(* IEC 61131-3 sources: actuators/test, 15 files *)

(* ---- Await.st ---- *)
USING AxUnit.Assert;
USING Simatic.Ax.Commands;

NAMESPACE Simatic.Ax.Actuators

    // Helper function to await the completion of a command and return its state.
    FUNCTION Await : PlcOpen
        VAR_INPUT
            cmd : itfCommand;
        END_VAR

        IF (NOT cmd.Busy()) THEN
            IF cmd.Done() THEN
                Await := PlcOpen#Done;
                RETURN;
            ELSIF cmd.Error() THEN
                Await := PlcOpen#Error;
                RETURN;
            ELSIF cmd.CommandAborted() THEN
                Await := PlcOpen#Aborted;
                RETURN;
            ELSE
                Await := PlcOpen#Undefined;
                RETURN;
            END_IF;
        ELSE
            Await := PlcOpen#Busy;
            RETURN;
        END_IF;
    END_FUNCTION

    // Enumeration representing the possible states of a PLCOpen command.
    TYPE
        PlcOpen : (Busy, Done, Error, Aborted, Undefined) := Undefined;
    END_TYPE

END_NAMESPACE

(* ---- ActuatorStateAssertions.st ---- *)
USING System.Strings;
USING AxUnit.ResultFunctions;
USING Simatic.Ax.Actuators;

NAMESPACE AxUnit.Assert

    FUNCTION Equal
        VAR_INPUT
            expected : ActuatorState;
            actual : ActuatorState;
            {CallerFilePath}
            file : WSTRING[1024];
            {CallerLineNumber}
            line : INT;
        END_VAR
        VAR_TEMP
            messageStr : STRING;
        END_VAR

        IF expected = actual THEN
            axunit_Succeed();
        ELSE
            messageStr := Concat('Expected = ', Simatic.Ax.Actuators.ToString(val := expected), ' Actual = ', Simatic.Ax.Actuators.ToString(actual));
            axunit_Fail(messageStr, file, line);
        END_IF;
        AxUnit.Assert.Equal(expected := TRUE, actual := expected = actual);
        ;
    END_FUNCTION

    FUNCTION NotEqual
        VAR_INPUT
            expected : ActuatorState;
            actual : ActuatorState;
            {CallerFilePath}
            file : WSTRING[1024];
            {CallerLineNumber}
            line : INT;
        END_VAR
        VAR_TEMP
            messageStr : STRING;
        END_VAR
        IF expected = actual THEN
            axunit_Succeed();
        ELSE
            messageStr := Concat('Expected = ', Simatic.Ax.Actuators.ToString(expected), 'Actual = ', Simatic.Ax.Actuators.ToString(actual));
            axunit_Fail(messageStr, file, line);
        END_IF;
        AxUnit.Assert.Equal(expected := TRUE, actual := expected <> actual);
        ;
    END_FUNCTION

END_NAMESPACE

(* ---- Asserts.st ---- *)
USING System.Strings;
USING AxUnit.ResultFunctions;

NAMESPACE AxUnit.Assert

    FUNCTION Equal
        VAR_INPUT
            expected : STRING;
            actual : STRING;
            {CallerFilePath}
            file : WSTRING[1024];
            {CallerLineNumber}
            line : INT;
        END_VAR
        VAR_TEMP
            messageStr : STRING;
        END_VAR

        IF expected = actual THEN
            axunit_Succeed();
        ELSE
            messageStr := Concat('Expected = ', expected, 'Actual = ', actual);
            axunit_Fail(messageStr, file, line);
        END_IF;
        Equal(expected := TRUE, actual := expected = actual);
        ;
    END_FUNCTION

    FUNCTION NotEqual
        VAR_INPUT
            expected : STRING;
            actual : STRING;
            {CallerFilePath}
            file : WSTRING[1024];
            {CallerLineNumber}
            line : INT;
        END_VAR
        VAR_TEMP
            messageStr : STRING;
        END_VAR

        IF expected = actual THEN
            axunit_Succeed();
        ELSE
            messageStr := Concat('Expected = ', expected, 'Actual = ', actual);
            axunit_Fail(messageStr, file, line);
        END_IF;
        Equal(expected := TRUE, actual := expected <> actual);
        ;
    END_FUNCTION

END_NAMESPACE

(* ---- Boolean.st ---- *)
USING AxUnit.ResultFunctions;
USING System.Strings;

NAMESPACE AxUnit.Assert

    FUNCTION PUBLIC IsTrue
        VAR_INPUT
            condition : BOOL;

            {CallerFilePath}
            file : WSTRING[1024];
            {CallerLineNumber}
            line : INT;
        END_VAR

        IF condition THEN
            axunit_Succeed();
        ELSE
            axunit_Fail('Condition is not true', file, line);
        END_IF;

    END_FUNCTION

    FUNCTION PUBLIC IsFalse
        VAR_INPUT
            condition : BOOL;

            {CallerFilePath}
            file : WSTRING[1024];
            {CallerLineNumber}
            line : INT;
        END_VAR

        IF NOT condition THEN
            axunit_Succeed();
        ELSE
            axunit_Fail('Condition is not false', file, line);
        END_IF;

    END_FUNCTION

END_NAMESPACE

(* ---- PlcOpenAssert.st ---- *)
USING Simatic.Ax.Commands;
USING System.Strings;
USING AxUnit.ResultFunctions;

NAMESPACE AxUnit.Assert

    FUNCTION Equal
        VAR_INPUT
            expected : PlcOpen;
            actual : PlcOpen;
            {CallerFilePath}
            file : WSTRING[1024];
            {CallerLineNumber}
            line : INT;
        END_VAR
        VAR_TEMP
            messageStr : STRING;
        END_VAR

        IF expected = actual THEN
            axunit_Succeed();
        ELSE
            messageStr := Concat('Expected = ', ToString(expected), 'Actual = ', ToString(actual));
            axunit_Fail(messageStr, file, line);
        END_IF;
        Equal(expected := TRUE, actual := expected = actual);
        ;
    END_FUNCTION

    FUNCTION NotEqual
        VAR_INPUT
            expected : PlcOpen;
            actual : PlcOpen;
            {CallerFilePath}
            file : WSTRING[1024];
            {CallerLineNumber}
            line : INT;
        END_VAR
        VAR_TEMP
            messageStr : STRING;
        END_VAR

        IF expected = actual THEN
            axunit_Succeed();
        ELSE
            messageStr := Concat('Expected = ', ToString(expected), ' Actual = ', ToString(actual));
            axunit_Fail(messageStr, file, line);
        END_IF;
        Equal(expected := TRUE, actual := expected <> actual);
        ;
    END_FUNCTION

END_NAMESPACE

(* ---- EndSwitchMock.st ---- *)
USING AxUnit.Assert;

NAMESPACE Simatic.Ax.Actuators

    /// Mock implementation of an activated endswitch for testing purposes.
    /// Input: None.
    /// Returns: Always returns TRUE for IsActivated, FALSE for all other state queries.
    CLASS EndSwitchMockActivated IMPLEMENTS itfEndswitch

        /// Starts monitoring the endswitch with a specified monitoring time.
        /// Input: Mode - The supervision mode to enable.
        /// Returns: None.
        METHOD PUBLIC EnableSupervision
            VAR_INPUT
                Mode : SuperVisionMode;
            END_VAR

            ;
        END_METHOD

        /// Checks if the endswitch is currently activated.
        /// Input: None.
        /// Returns: Always TRUE to simulate an activated endswitch.
        METHOD PUBLIC IsActivated : BOOL
            IsActivated := TRUE;
            ;
        END_METHOD

        /// Checks if the endswitch has been reached.
        /// Input: None.
        /// Returns: Always FALSE for this mock.
        METHOD PUBLIC HasReached : BOOL
            HasReached := FALSE;
            ;
        END_METHOD

        /// Checks if the endswitch has been left.
        /// Input: None.
        /// Returns: Always FALSE for this mock.
        METHOD PUBLIC HasLeft : BOOL
            HasLeft := FALSE;
            ;
        END_METHOD

        /// Checks if the monitoring time has elapsed.
        /// Input: None.
        /// Returns: Always FALSE for this mock.
        METHOD PUBLIC TimeHasElapsed : BOOL
            TimeHasElapsed := FALSE;
        END_METHOD

        /// Returns the error status of the endswitch.
        /// Input: None.
        /// Returns: Default supervision error state.
        METHOD PUBLIC GetError : SuperVisionState
            ;
        END_METHOD
    END_CLASS

    /// Mock implementation of an endswitch that has been reached for testing purposes.
    /// Input: None.
    /// Returns: TRUE for IsActivated and HasReached, FALSE for other state queries.
    CLASS EndSwitchMockHasReached IMPLEMENTS itfEndswitch

        /// Starts monitoring the endswitch with a specified monitoring time.
        /// Input: Mode - The supervision mode to enable.
        /// Returns: None.
        METHOD PUBLIC EnableSupervision
            VAR_INPUT
                Mode : SuperVisionMode;
            END_VAR
            ;
        END_METHOD

        /// Checks if the endswitch is currently activated.
        /// Input: None.
        /// Returns: Always TRUE to simulate an activated endswitch.
        METHOD PUBLIC IsActivated : BOOL
            IsActivated := TRUE;
            ;
        END_METHOD

        /// Checks if the endswitch has been reached.
        /// Input: None.
        /// Returns: Always TRUE to simulate a reached endswitch.
        METHOD PUBLIC HasReached : BOOL
            HasReached := TRUE;
            ;
        END_METHOD

        /// Checks if the endswitch has been left.
        /// Input: None.
        /// Returns: Always FALSE for this mock.
        METHOD PUBLIC HasLeft : BOOL
            HasLeft := FALSE;
            ;
        END_METHOD

        /// Checks if the monitoring time has elapsed.
        /// Input: None.
        /// Returns: Always FALSE for this mock.
        METHOD PUBLIC TimeHasElapsed : BOOL
            TimeHasElapsed := FALSE;
        END_METHOD

        /// Returns the error status of the endswitch.
        /// Input: None.
        /// Returns: Default supervision error state.
        METHOD PUBLIC GetError : SuperVisionState
            ;
        END_METHOD
    END_CLASS

    /// Mock implementation of an endswitch that has been left for testing purposes.
    /// Input: None.
    /// Returns: TRUE for HasLeft, FALSE for other state queries.
    CLASS EndSwitchMockHasLeft IMPLEMENTS itfEndswitch

        /// Starts monitoring the endswitch with a specified monitoring time.
        /// Input: Mode - The supervision mode to enable.
        /// Returns: None.
        METHOD PUBLIC EnableSupervision
            VAR_INPUT
                Mode : SuperVisionMode;
            END_VAR

            ;
        END_METHOD

        /// Checks if the endswitch is currently activated.
        /// Input: None.
        /// Returns: Always FALSE to simulate a deactivated endswitch.
        METHOD PUBLIC IsActivated : BOOL
            IsActivated := FALSE;
            ;
        END_METHOD

        /// Checks if the endswitch has been reached.
        /// Input: None.
        /// Returns: Always FALSE for this mock.
        METHOD PUBLIC HasReached : BOOL
            HasReached := FALSE;
            ;
        END_METHOD

        /// Checks if the endswitch has been left.
        /// Input: None.
        /// Returns: Always TRUE to simulate a left endswitch.
        METHOD PUBLIC HasLeft : BOOL
            HasLeft := TRUE;
            ;
        END_METHOD

        /// Checks if the monitoring time has elapsed.
        /// Input: None.
        /// Returns: Always FALSE for this mock.
        METHOD PUBLIC TimeHasElapsed : BOOL
            TimeHasElapsed := FALSE;
        END_METHOD

        /// Returns the error status of the endswitch.
        /// Input: None.
        /// Returns: Default supervision error state.
        METHOD PUBLIC GetError : SuperVisionState
            ;
        END_METHOD
    END_CLASS

    /// Mock implementation of a non-activated endswitch for testing purposes.
    /// Input: None.
    /// Returns: FALSE for all state queries to simulate an inactive endswitch.
    CLASS EndSwitchMockNotActivated IMPLEMENTS itfEndswitch

        /// Starts monitoring the endswitch with a specified monitoring time.
        /// Input: Mode - The supervision mode to enable.
        /// Returns: None.
        METHOD PUBLIC EnableSupervision
            VAR_INPUT
                Mode : SuperVisionMode;
            END_VAR

            ;
        END_METHOD

        /// Disables monitoring of the endswitch.
        /// Input: None.
        /// Returns: None.
        METHOD PUBLIC DisableMonitoring
            ;
        END_METHOD

        /// Checks if the endswitch is currently activated.
        /// Input: None.
        /// Returns: Always FALSE to simulate an inactive endswitch.
        METHOD PUBLIC IsActivated : BOOL
            IsActivated := FALSE;
            ;
        END_METHOD

        /// Checks if the endswitch has been reached.
        /// Input: None.
        /// Returns: Always FALSE for this mock.
        METHOD PUBLIC HasReached : BOOL
            HasReached := FALSE;
            ;
        END_METHOD

        /// Checks if the endswitch has been left.
        /// Input: None.
        /// Returns: Always FALSE for this mock.
        METHOD PUBLIC HasLeft : BOOL
            HasLeft := FALSE;
            ;
        END_METHOD

        /// Checks if the monitoring time has elapsed.
        /// Input: None.
        /// Returns: Always FALSE for this mock.
        METHOD PUBLIC TimeHasElapsed : BOOL
            TimeHasElapsed := FALSE;
        END_METHOD

        /// Returns the error status of the endswitch.
        /// Input: None.
        /// Returns: Default supervision error state.
        METHOD PUBLIC GetError : SuperVisionState
            ;
        END_METHOD
    END_CLASS
END_NAMESPACE

(* ---- TestActuator2Way.st ---- *)
USING AxUnit.Assert;
USING Simatic.Ax.Commands;

NAMESPACE Simatic.Ax.Actuators

    {TestFixture}
    // Test class for the Actuator2Way class.
    // This class contains tests to verify the behavior of the Actuator2Way component.
    CLASS TestActuator2Way
        VAR
            // Instance of Actuator2Way for testing.
            _actuator, _actuatorStateless : Actuator2Way;

            // Command interface for actuator operations.
            _cmd : itfCommand;

            // State of the PLCOpen command.
            _plcOpenState : PlcOpen;

            // Mock sensors for testing actuator behavior.
            _sensorActivated : EndSwitchMockActivated;
            _sensorNotActivated : EndSwitchMockNotActivated;
            _sensorHasReached : EndSwitchMockHasReached;
            _sensorHasLeft : EndSwitchMockHasLeft;

            // Actuator Controls
            ActuatorMoveToHomePos : PositionControl;
            ActuatorMoveToWorkPos : PositionControl;
        END_VAR

        {TestSetup}
        // Sets up the test environment by initializing the actuator instance and assigning mock sensors and controls.
        METHOD PUBLIC Setup
            _actuator := _actuatorStateless;
            _actuator.Q_ToHomePosition := ActuatorMoveToHomePos;
            _actuator.Q_ToWorkPosition := ActuatorMoveToWorkPos;
        END_METHOD

        {Test}
        // Verifies that the initial state of the actuator is Undefined.
        METHOD PUBLIC TestInitialState
            VAR
                initialState : ActuatorState;
            END_VAR

            // Step 1: Retrieve the initial state of the actuator.
            initialState := _actuator.GetState();

            // Step 2: Assert that the initial state is Undefined.
            Equal(expected := ActuatorState#Undefined, actual := initialState);
        END_METHOD

        {Test}
        // Tests the transition to MoveToWorkPosition state when not in the work position.
        METHOD PUBLIC Command_MoveToWorkPosition_Returns_State_MoveToWorkPosition_When_NotInWorkpos
            VAR
                resultHome, resultWork : BOOL;
            END_VAR

            // Step 1: Set initial sensor states to indicate the actuator is not in any position.
            _actuator.I_InHomePosition := _sensorNotActivated;
            _actuator.I_InWorkPosition := _sensorNotActivated;

            // Step 2: Issue the command to move to work position.
            _cmd := _actuator.GoToWorkPosition();
            _plcOpenState := Await(_cmd);

            // Step 3: Verify the actuator is in the MoveToWorkPosition state.
            Equal(expected := PlcOpen#Busy, actual := _plcOpenState);
            Equal(expected := ActuatorState#MoveToWorkPosition, actual := _actuator.GetState());

            // Step 4: Check the actuator outputs.
            ActuatorMoveToHomePos.WriteCyclic(Q => resultHome);
            ActuatorMoveToWorkPos.WriteCyclic(Q => resultWork);
            IsFalse(condition := resultHome);
            IsTrue(condition := resultWork);

            // Step 5: Simulate reaching the work position.
            _actuator.I_InWorkPosition := _sensorHasReached;
            _plcOpenState := Await(_cmd);

            // Step 6: Verify the actuator has reached the work position.
            Equal(expected := PlcOpen#Done, actual := _plcOpenState);
            Equal(expected := ActuatorState#InWorkPosition, actual := _actuator.GetState());

            // Step 7: Check the actuator outputs again.
            ActuatorMoveToHomePos.WriteCyclic(Q => resultHome);
            ActuatorMoveToWorkPos.WriteCyclic(Q => resultWork);
            IsFalse(condition := resultHome);
            IsFalse(condition := resultWork);
        END_METHOD

        {Test}
        // Tests that the actuator remains in InWorkPosition state when already in the work position.
        METHOD PUBLIC Command_MoveToWorkPosition_Returns_State_InWorkPosition_When_InWorkpos
            VAR
                isInWorkPos : BOOL := TRUE;
            END_VAR

            // Step 1: Set initial sensor states to indicate the actuator is already in the work position.
            _actuator.I_InHomePosition := _sensorNotActivated;
            _actuator.I_InWorkPosition := _sensorActivated;

            // Step 2: Issue the command to move to work position.
            _cmd := _actuator.GoToWorkPosition();
            _plcOpenState := Await(_cmd);

            // Step 3: Verify the actuator remains in the InWorkPosition state.
            Equal(expected := PlcOpen#Done, actual := _plcOpenState);
            Equal(expected := ActuatorState#InWorkPosition, actual := _actuator.GetState());
        END_METHOD

        {Test}
        // Tests the transition to MoveToHomePosition state when not in the home position.
        METHOD PUBLIC Command_MoveToHomePosition_Returns_State_MoveToHomePosition_When_NotIn_HomePos
            VAR
                resultHome, resultWork : BOOL;
            END_VAR

            // Step 1: Set initial sensor states to indicate the actuator is not in any position.
            _actuator.I_InHomePosition := _sensorNotActivated;
            _actuator.I_InWorkPosition := _sensorNotActivated;

            // Step 2: Issue the command to move to home position.
            _cmd := _actuator.GoToHomePosition();
            _plcOpenState := Await(_cmd);

            // Step 3: Verify the actuator is in the MoveToHomePosition state.
            Equal(expected := PlcOpen#Busy, actual := _plcOpenState);
            Equal(expected := ActuatorState#MoveToHomePosition, actual := _actuator.GetState());

            // Step 4: Check the actuator outputs.
            ActuatorMoveToHomePos.WriteCyclic(Q => resultHome);
            ActuatorMoveToWorkPos.WriteCyclic(Q => resultWork);
            IsTrue(condition := resultHome);
            IsFalse(condition := resultWork);

            // Step 5: Simulate reaching the home position.
            _actuator.I_InHomePosition := _sensorHasReached;
            _plcOpenState := Await(_cmd);

            // Step 6: Verify the actuator has reached the home position.
            Equal(expected := PlcOpen#Done, actual := _plcOpenState);
            Equal(expected := ActuatorState#InHomePosition, actual := _actuator.GetState());

            // Step 7: Check the actuator outputs again.
            ActuatorMoveToHomePos.WriteCyclic(Q => resultHome);
            ActuatorMoveToWorkPos.WriteCyclic(Q => resultWork);
            IsFalse(condition := resultHome);
            IsFalse(condition := resultWork);
        END_METHOD

        {Test}
        // Tests that the actuator remains in InHomePosition state when already in the home position.
        METHOD PUBLIC Command_MoveToHomePosition_Returns_State_InHomePosition_When_In_HomePos
            VAR
                isInHomePos : BOOL := TRUE;
            END_VAR

            // Step 1: Set initial sensor states to indicate the actuator is already in the home position.
            _actuator.I_InHomePosition := _sensorActivated;
            _actuator.I_InWorkPosition := _sensorNotActivated;

            // Step 2: Issue the command to move to home position.
            _cmd := _actuator.GoToHomePosition();
            _plcOpenState := Await(_cmd);

            // Step 3: Verify the actuator remains in the InHomePosition state.
            Equal(expected := PlcOpen#Done, actual := _plcOpenState);
            Equal(expected := ActuatorState#InHomePosition, actual := _actuator.GetState());
        END_METHOD

        {Test}
        // Tests multiple calls to the MoveToWorkPosition command.
        METHOD PUBLIC Call_Command_MoveToWorkPosition_Multiple
            VAR
                isInHomePos : BOOL := TRUE;
            END_VAR

            // Step 1: Set initial sensor states to indicate the actuator is not in any position.
            _actuator.I_InHomePosition := _sensorNotActivated;
            _actuator.I_InWorkPosition := _sensorNotActivated;

            // Step 2: Issue the command to move to work position multiple times.
            _cmd := _actuator.GoToWorkPosition();
            _plcOpenState := Await(_cmd);
            Equal(expected := PlcOpen#Busy, actual := _plcOpenState);
            Equal(expected := ActuatorState#MoveToWorkPosition, actual := _actuator.GetState());

            _cmd := _actuator.GoToWorkPosition();
            _plcOpenState := Await(_cmd);
            Equal(expected := PlcOpen#Busy, actual := _plcOpenState);
            Equal(expected := ActuatorState#MoveToWorkPosition, actual := _actuator.GetState());

            _cmd := _actuator.GoToWorkPosition();
            _plcOpenState := Await(_cmd);
            Equal(expected := PlcOpen#Busy, actual := _plcOpenState);
            Equal(expected := ActuatorState#MoveToWorkPosition, actual := _actuator.GetState());

            // Step 3: Simulate reaching the work position.
            _actuator.I_InWorkPosition := _sensorActivated;
            _cmd := _actuator.GoToWorkPosition();
            Equal(expected := ActuatorState#InWorkPosition, actual := _actuator.GetState());
            _plcOpenState := Await(_cmd);
            Equal(expected := PlcOpen#Done, actual := _plcOpenState);
            Equal(expected := ActuatorState#InWorkPosition, actual := _actuator.GetState());
        END_METHOD

        {Test}
        // Tests the behavior when MoveToWorkPosition is interrupted by MoveToHomePosition.
        METHOD PUBLIC Command_MoveToWorkPosition_Interrupted_By_MoveToHomePosition
            VAR
                resultHome, resultWork : BOOL;
            END_VAR

            // Step 1: Set initial sensor states to indicate the actuator is not in any position.
            _actuator.I_InHomePosition := _sensorNotActivated;
            _actuator.I_InWorkPosition := _sensorNotActivated;

            // Step 2: Start MoveToWorkPosition.
            _cmd := _actuator.GoToWorkPosition();
            _plcOpenState := Await(_cmd);

            // Step 3: Verify the actuator is in the MoveToWorkPosition state.
            Equal(expected := PlcOpen#Busy, actual := _plcOpenState);
            Equal(expected := ActuatorState#MoveToWorkPosition, actual := _actuator.GetState());

            // Step 4: Check the actuator outputs.
            ActuatorMoveToHomePos.WriteCyclic(Q => resultHome);
            ActuatorMoveToWorkPos.WriteCyclic(Q => resultWork);
            IsFalse(condition := resultHome);
            IsTrue(condition := resultWork);

            // Step 5: Interrupt with MoveToHomePosition.
            _cmd := _actuator.GoToHomePosition();
            _plcOpenState := Await(_cmd);

            // Step 6: Verify the actuator is in the MoveToHomePosition state.
            Equal(expected := PlcOpen#Busy, actual := _plcOpenState);
            Equal(expected := ActuatorState#MoveToHomePosition, actual := _actuator.GetState());

            // Step 7: Check the actuator outputs.
            ActuatorMoveToHomePos.WriteCyclic(Q => resultHome);
            ActuatorMoveToWorkPos.WriteCyclic(Q => resultWork);
            IsTrue(condition := resultHome);
            IsFalse(condition := resultWork);

            // Step 8: Simulate reaching the home position.
            _actuator.I_InHomePosition := _sensorHasReached;
            _plcOpenState := Await(_cmd);

            // Step 9: Verify the actuator has reached the home position.
            Equal(expected := PlcOpen#Done, actual := _plcOpenState);
            Equal(expected := ActuatorState#InHomePosition, actual := _actuator.GetState());

            // Step 10: Check the actuator outputs again.
            ActuatorMoveToHomePos.WriteCyclic(Q => resultHome);
            ActuatorMoveToWorkPos.WriteCyclic(Q => resultWork);
            IsFalse(condition := resultHome);
            IsFalse(condition := resultWork);
        END_METHOD

        {Test}
        // Tests the behavior when MoveToHomePosition is interrupted by MoveToWorkPosition.
        METHOD PUBLIC Command_MoveToHomePosition_Interrupted_By_MoveToWorkPosition
            VAR
                resultHome, resultWork : BOOL;
            END_VAR

            // Step 1: Set initial sensor states to indicate the actuator is not in any position.
            _actuator.I_InHomePosition := _sensorNotActivated;
            _actuator.I_InWorkPosition := _sensorNotActivated;

            // Step 2: Start MoveToHomePosition.
            _cmd := _actuator.GoToHomePosition();
            _plcOpenState := Await(_cmd);

            // Step 3: Verify the actuator is in the MoveToHomePosition state.
            Equal(expected := PlcOpen#Busy, actual := _plcOpenState);
            Equal(expected := ActuatorState#MoveToHomePosition, actual := _actuator.GetState());

            // Step 4: Check the actuator outputs.
            ActuatorMoveToHomePos.WriteCyclic(Q => resultHome);
            ActuatorMoveToWorkPos.WriteCyclic(Q => resultWork);
            IsTrue(condition := resultHome);
            IsFalse(condition := resultWork);

            // Step 5: Interrupt with MoveToWorkPosition.
            _cmd := _actuator.GoToWorkPosition();
            _plcOpenState := Await(_cmd);

            // Step 6: Verify the actuator is in the MoveToWorkPosition state.
            Equal(expected := PlcOpen#Busy, actual := _plcOpenState);
            Equal(expected := ActuatorState#MoveToWorkPosition, actual := _actuator.GetState());

            // Step 7: Check the actuator outputs.
            ActuatorMoveToHomePos.WriteCyclic(Q => resultHome);
            ActuatorMoveToWorkPos.WriteCyclic(Q => resultWork);
            IsFalse(condition := resultHome);
            IsTrue(condition := resultWork);

            // Step 8: Simulate reaching the work position.
            _actuator.I_InWorkPosition := _sensorHasReached;
            _plcOpenState := Await(_cmd);

            // Step 9: Verify the actuator has reached the work position.
            Equal(expected := PlcOpen#Done, actual := _plcOpenState);
            Equal(expected := ActuatorState#InWorkPosition, actual := _actuator.GetState());

            // Step 10: Check the actuator outputs again.
            ActuatorMoveToHomePos.WriteCyclic(Q => resultHome);
            ActuatorMoveToWorkPos.WriteCyclic(Q => resultWork);
            IsFalse(condition := resultHome);
            IsFalse(condition := resultWork);
        END_METHOD
    END_CLASS

END_NAMESPACE

(* ---- TestActuator2WayErrorHandling.st ---- *)
USING AxUnit.Assert;
USING Simatic.Ax.Commands;

NAMESPACE Simatic.Ax.Actuators

    {TestFixture}
    // Test class for the Actuator2Way class.
    // This class contains tests to verify the behavior of the Actuator2Way component.
    CLASS TestActuator2WayErrorHandling
        VAR
            // Instance of Actuator2Way for testing.
            _actuator, _actuatorStateless : Actuator2Way;

            // Command interface for actuator operations.
            _cmd : itfCommand;

            // State of the PLCOpen command.
            _plcOpenState : PlcOpen;

            // Mock sensors for testing actuator behavior.
            _sensorActivated : EndSwitchMockActivated;
            _sensorNotActivated : EndSwitchMockNotActivated;
            _sensorHasReached : EndSwitchMockHasReached;
            _sensorHasLeft : EndSwitchMockHasLeft;
            _sensorTimeHasElapsed : EndSwitchMockTimeHasElapsed;

            // Actuator Controls
            ActuatorMoveToHomePos : PositionControl;
            ActuatorMoveToWorkPos : PositionControl;
        END_VAR

        {TestSetup}
        // Sets up the test environment by initializing the actuator instance and assigning mock sensors and controls.
        METHOD PUBLIC Setup
            _actuator := _actuatorStateless;
            _actuator.Q_ToHomePosition := ActuatorMoveToHomePos;
            _actuator.Q_ToWorkPosition := ActuatorMoveToWorkPos;
            _actuator.I_InWorkPosition := _sensorNotActivated;
            _actuator.I_InHomePosition := _sensorNotActivated;
        END_METHOD

        {Test}
        // Tests the transition to MoveToWorkPosition state when not in the work position.
        METHOD PUBLIC Command_MoveToWorkPosition_Error_When_Sensor_Time_Has_Elapsed
            VAR
                resultHome, resultWork : BOOL;
            END_VAR

            // Step 1: Set initial sensor states to indicate the actuator is not in any position.
            _actuator.I_InHomePosition := _sensorNotActivated;
            _actuator.I_InWorkPosition := _sensorNotActivated;

            // Step 2: Issue the command to move to work position.
            _cmd := _actuator.GoToWorkPosition();
            _plcOpenState := Await(_cmd);

            // Step 3: Verify the actuator is in the MoveToWorkPosition state.
            Equal(expected := PlcOpen#Busy, actual := _plcOpenState);
            Equal(expected := ActuatorState#MoveToWorkPosition, actual := _actuator.GetState());

            // Step 4: Check the actuator outputs.
            ActuatorMoveToHomePos.WriteCyclic(Q => resultHome);
            ActuatorMoveToWorkPos.WriteCyclic(Q => resultWork);
            IsFalse(condition := resultHome);
            IsTrue(condition := resultWork);

            // Step 5: Simulate reaching the work position.
            _actuator.I_InWorkPosition := _sensorTimeHasElapsed;
            _plcOpenState := Await(_cmd);

            // Step 6: Verify the actuator has reached the work position.
            Equal(expected := PlcOpen#Error, actual := _plcOpenState);
            Equal(expected := ActuatorState#Error, actual := _actuator.GetState());

            // Step 7: Check the actuator outputs again.
            ActuatorMoveToHomePos.WriteCyclic(Q => resultHome);
            ActuatorMoveToWorkPos.WriteCyclic(Q => resultWork);
            IsFalse(condition := resultHome);
            IsFalse(condition := resultWork);
        END_METHOD

        {Test}
        // Tests the transition to MoveToHomePosition state when not in the home position.
        METHOD PUBLIC Reset_Actuator_Returns
            VAR
                resultHome, resultWork : BOOL;
            END_VAR
            THIS.Command_MoveToWorkPosition_Error_When_Sensor_Time_Has_Elapsed();
            // Step 1: Reset Actuator

            _actuator.Reset();

            // Step 2: Verify the actuator is in the MoveToHomePosition state.
            Equal(expected := ActuatorState#Undefined, actual := _actuator.GetState());

            // Step 3: Check the actuator outputs again.
            ActuatorMoveToHomePos.WriteCyclic(Q => resultHome);
            ActuatorMoveToWorkPos.WriteCyclic(Q => resultWork);
            IsFalse(condition := resultHome);
            IsFalse(condition := resultWork);
        END_METHOD

        {Test}
        // Tests the transition to MoveToWorkPosition state when not in the work position.
        METHOD PUBLIC Both_sensors_Active_Retrurs_Error
            VAR
                resultHome, resultWork : BOOL;
            END_VAR

            // Step 1: Set initial sensor states to indicate the actuator is not in any position.
            _actuator.I_InHomePosition := _sensorActivated;
            _actuator.I_InWorkPosition := _sensorActivated;

            // Step 2: Issue the command to move to work position.
            _cmd := _actuator.GoToWorkPosition();
            _plcOpenState := Await(_cmd);

            // Step 3: Verify the actuator is in the MoveToWorkPosition state.
            Equal(expected := PlcOpen#Error, actual := _plcOpenState);
            Equal(expected := ActuatorState#Error, actual := _actuator.GetState());

            // Step 4: Check the actuator outputs again.
            ActuatorMoveToHomePos.WriteCyclic(Q => resultHome);
            ActuatorMoveToWorkPos.WriteCyclic(Q => resultWork);
            IsFalse(condition := resultHome);
            IsFalse(condition := resultWork);
        END_METHOD
    END_CLASS

END_NAMESPACE

(* ---- TestActuator2WayWithLogger.st ---- *)
USING AxUnit.Assert;
USING Simatic.Ax.Commands;

NAMESPACE Simatic.Ax.Actuators

    {TestFixture}
    // Test class for the Actuator2Way class.
    // This class contains tests to verify the behavior of the Actuator2Way component.
    CLASS TestActuator2WayWithLogger
        VAR
            // Instance of Actuator2Way for testing.
            _actuator, _actuatorStateless : Actuator2Way;

            // Command interface for actuator operations.
            _cmd : itfCommand;

            // Logger
            _logger : StateLogger;
            _msgBuffer : ARRAY[1..1] OF LogMessage;

            // State of the PLCOpen command.
            _plcOpenState : PlcOpen;

            // Mock sensors for testing actuator behavior.
            _sensorActivated : EndSwitchMockActivated;
            _sensorNotActivated : EndSwitchMockNotActivated;
            _sensorHasReached : EndSwitchMockHasReached;
            _sensorHasLeft : EndSwitchMockHasLeft;

        END_VAR

        {TestSetup}
        // Sets up the test environment by initializing the actuator instance and assigning mock sensors and controls.
        METHOD PUBLIC Setup
            _actuator := _actuatorStateless;
            _actuator.Logger := _logger;
            _logger.MsgBuffer := REF(_msgBuffer);
            _logger.SetLogLevel(LogLevel#Info);
        END_METHOD

        {Test}
        // Tests the state transitions and verifies log entries in the StateLogger.
        METHOD PUBLIC Test_a_CompleteSequence_to_check_the_LogMessages
            VAR
                logEntry : STRING;
            END_VAR

            // Step 1: Set initial sensor states to indicate the actuator is in the home position.
            _actuator.I_InHomePosition := _sensorActivated;
            _actuator.I_InWorkPosition := _sensorNotActivated;

            // Step 2: Issue the command to move to work position.
            _cmd := _actuator.GoToWorkPosition();
            _plcOpenState := Await(_cmd);

            // Step 3: Verify the log entry for State changed to MoveToWorkPosition.
            logEntry := _logger.MsgBuffer^[1].message;
            Equal(expected := 'State changed to MoveToWorkPosition', actual := logEntry);

            // Step 4: Simulate reaching the work position.
            _actuator.I_InWorkPosition := _sensorHasReached;
            _actuator.I_InHomePosition := _sensorNotActivated;
            _plcOpenState := Await(_cmd);

            // Step 5: Verify the log entry for reaching InWorkPosition.
            logEntry := _logger.MsgBuffer^[1].message;
            Equal(expected := 'State changed to InWorkPosition', actual := logEntry);

            // Step 6: Issue the command to move to home position.
            _cmd := _actuator.GoToHomePosition();
            _plcOpenState := Await(_cmd);

            // Step 7: Verify the log entry for State changed to MoveToHomePosition.
            logEntry := _logger.MsgBuffer^[1].message;
            Equal(expected := 'State changed to MoveToHomePosition', actual := logEntry);

            // Step 8: Simulate reaching the home position.
            _actuator.I_InHomePosition := _sensorHasReached;
            _plcOpenState := Await(_cmd);

            // Step 9: Verify the log entry for reaching InHomePosition.
            logEntry := _logger.MsgBuffer^[1].message;
            Equal(expected := 'State changed to InHomePosition', actual := logEntry);
        END_METHOD

    END_CLASS

END_NAMESPACE

(* ---- TestActuator3Way.st ---- *)
USING AxUnit.Assert;
USING Simatic.Ax.Commands;

NAMESPACE Simatic.Ax.Actuators

    {TestFixture}
    // Test class for the Actuator3Way class.
    // This class contains tests to verify the behavior of the Actuator3Way component.
    CLASS TestActuator3Way
        VAR
            // Instance of Actuator3Way for testing.
            _actuator, _actuatorStateless : Actuator3Way;

            // Command interface for actuator operations.
            _cmd : itfCommand;

            // State of the PLCOpen command.
            _plcOpenState : PlcOpen;

            // Mock sensors for testing actuator behavior.
            _sensorActivated : EndSwitchMockActivated;
            _sensorNotActivated : EndSwitchMockNotActivated;
            _sensorHasReached : EndSwitchMockHasReached;
            _sensorHasLeft : EndSwitchMockHasLeft;

            // Actuator Controls
            ActuatorMoveToHomePos : PositionControl;
            ActuatorMoveToWorkPos : PositionControl;
            ActuatorMoveToWorkPos2 : PositionControl;
        END_VAR

        {TestSetup}
        // Sets up the test environment by initializing the actuator instance and assigning mock sensors and controls.
        METHOD PUBLIC Setup
            _actuator := _actuatorStateless;
            _actuator.Q_ToHomePosition := ActuatorMoveToHomePos;
            _actuator.Q_ToWorkPosition := ActuatorMoveToWorkPos;
            _actuator.Q_ToWorkPosition2 := ActuatorMoveToWorkPos2;
        END_METHOD

        {Test}
        // Verifies that the initial state of the actuator is Undefined.
        METHOD PUBLIC TestInitialState
            VAR
                initialState : ActuatorState;
            END_VAR

            // Step 1: Retrieve the initial state of the actuator.
            initialState := _actuator.GetState();

            // Step 2: Assert that the initial state is Undefined.
            Equal(expected := ActuatorState#Undefined, actual := initialState);
        END_METHOD

        {Test}
        // Tests the transition to MoveToWorkPosition state when not in the work position.
        METHOD PUBLIC Command_MoveToWorkPosition_Returns_State_MoveToWorkPosition_When_NotInWorkpos
            VAR
                resultHome, resultWork, resultWork2 : BOOL;
            END_VAR

            // Step 1: Set initial sensor states to indicate the actuator is not in any position.
            _actuator.I_InHomePosition := _sensorNotActivated;
            _actuator.I_InWorkPosition := _sensorNotActivated;
            _actuator.I_InWorkPosition2 := _sensorNotActivated;

            // Step 2: Issue the command to move to work position.
            _cmd := _actuator.GoToWorkPosition();
            _plcOpenState := Await(_cmd);

            // Step 3: Verify the actuator is in the MoveToWorkPosition state.
            AxUnit.Assert.Equal(expected := PlcOpen#Busy, actual := _plcOpenState);
            Equal(expected := ActuatorState#MoveToWorkPosition, actual := _actuator.GetState());

            // Step 4: Check the actuator outputs.
            ActuatorMoveToHomePos.WriteCyclic(Q => resultHome);
            ActuatorMoveToWorkPos.WriteCyclic(Q => resultWork);
            ActuatorMoveToWorkPos2.WriteCyclic(Q => resultWork2);
            IsFalse(condition := resultHome);
            IsTrue(condition := resultWork);
            IsFalse(condition := resultWork2);

            // Step 5: Simulate reaching the work position.
            _actuator.I_InWorkPosition := _sensorHasReached;
            _plcOpenState := Await(_cmd);

            // Step 6: Verify the actuator has reached the work position.
            AxUnit.Assert.Equal(expected := PlcOpen#Done, actual := _plcOpenState);
            Equal(expected := ActuatorState#InWorkPosition, actual := _actuator.GetState());

            // Step 7: Check the actuator outputs again.
            ActuatorMoveToHomePos.WriteCyclic(Q => resultHome);
            ActuatorMoveToWorkPos.WriteCyclic(Q => resultWork);
            ActuatorMoveToWorkPos2.WriteCyclic(Q => resultWork2);
            IsFalse(condition := resultHome);
            IsFalse(condition := resultWork);
            IsFalse(condition := resultWork2);
        END_METHOD

        {Test}
        // Tests the transition to MoveToWorkPosition2 state when not in the second work position.
        METHOD PUBLIC Command_MoveToWorkPosition2_Returns_State_MoveToWorkPosition2_When_NotInWorkpos2
            VAR
                resultHome, resultWork, resultWork2 : BOOL;
            END_VAR

            // Step 1: Set initial sensor states to indicate the actuator is not in any position.
            _actuator.I_InHomePosition := _sensorNotActivated;
            _actuator.I_InWorkPosition := _sensorNotActivated;
            _actuator.I_InWorkPosition2 := _sensorNotActivated;

            // Step 2: Issue the command to move to work position 2.
            _cmd := _actuator.GoToWorkPosition2();
            _plcOpenState := Await(_cmd);

            // Step 3: Verify the actuator is in the MoveToWorkPosition2 state.
            AxUnit.Assert.Equal(expected := PlcOpen#Busy, actual := _plcOpenState);
            Equal(expected := ActuatorState#MoveToWorkPosition2, actual := _actuator.GetState());

            // Step 4: Check the actuator outputs.
            ActuatorMoveToHomePos.WriteCyclic(Q => resultHome);
            ActuatorMoveToWorkPos.WriteCyclic(Q => resultWork);
            ActuatorMoveToWorkPos2.WriteCyclic(Q => resultWork2);
            IsFalse(condition := resultHome);
            IsFalse(condition := resultWork);
            IsTrue(condition := resultWork2);

            // Step 5: Simulate reaching the second work position.
            _actuator.I_InWorkPosition2 := _sensorHasReached;
            _plcOpenState := Await(_cmd);

            // Step 6: Verify the actuator has reached the second work position.
            AxUnit.Assert.Equal(expected := PlcOpen#Done, actual := _plcOpenState);
            Equal(expected := ActuatorState#InWorkPosition2, actual := _actuator.GetState());

            // Step 7: Check the actuator outputs again.
            ActuatorMoveToHomePos.WriteCyclic(Q => resultHome);
            ActuatorMoveToWorkPos.WriteCyclic(Q => resultWork);
            ActuatorMoveToWorkPos2.WriteCyclic(Q => resultWork2);
            IsFalse(condition := resultHome);
            IsFalse(condition := resultWork);
            IsFalse(condition := resultWork2);
        END_METHOD

        {Test}
        // Tests the transition to MoveToHomePosition state when not in the home position.
        METHOD PUBLIC Command_MoveToHomePosition_Returns_State_MoveToHomePosition_When_NotInHomePos
            VAR
                resultHome, resultWork, resultWork2 : BOOL;
            END_VAR

            // Step 1: Set initial sensor states to indicate the actuator is not in any position.
            _actuator.I_InHomePosition := _sensorNotActivated;
            _actuator.I_InWorkPosition := _sensorNotActivated;
            _actuator.I_InWorkPosition2 := _sensorNotActivated;

            // Step 2: Issue the command to move to home position.
            _cmd := _actuator.GoToHomePosition();
            _plcOpenState := Await(_cmd);

            // Step 3: Verify the actuator is in the MoveToHomePosition state.
            AxUnit.Assert.Equal(expected := PlcOpen#Busy, actual := _plcOpenState);
            Equal(expected := ActuatorState#MoveToHomePosition, actual := _actuator.GetState());

            // Step 4: Check the actuator outputs.
            ActuatorMoveToHomePos.WriteCyclic(Q => resultHome);
            ActuatorMoveToWorkPos.WriteCyclic(Q => resultWork);
            ActuatorMoveToWorkPos2.WriteCyclic(Q => resultWork2);
            IsTrue(condition := resultHome);
            IsFalse(condition := resultWork);
            IsFalse(condition := resultWork2);

            // Step 5: Simulate reaching the home position.
            _actuator.I_InHomePosition := _sensorHasReached;
            _plcOpenState := Await(_cmd);
            AxUnit.Assert.Equal(expected := PlcOpen#Done, actual := _plcOpenState);
            Equal(expected := ActuatorState#InHomePosition, actual := _actuator.GetState());

            ActuatorMoveToHomePos.WriteCyclic(Q => resultHome);
            ActuatorMoveToWorkPos.WriteCyclic(Q => resultWork);
            ActuatorMoveToWorkPos2.WriteCyclic(Q => resultWork2);
            IsFalse(condition := resultHome);
            IsFalse(condition := resultWork);
            IsFalse(condition := resultWork2);
        END_METHOD

        {Test}
        METHOD PUBLIC Call_Command_MoveToWorkPosition2_Multiple
            VAR
                isInHomePos : BOOL := TRUE;
            END_VAR

            _actuator.I_InHomePosition := _sensorNotActivated;
            _actuator.I_InWorkPosition := _sensorNotActivated;
            _actuator.I_InWorkPosition2 := _sensorNotActivated;

            _cmd := _actuator.GoToWorkPosition2();
            _plcOpenState := Await(_cmd);
            AxUnit.Assert.Equal(expected := PlcOpen#Busy, actual := _plcOpenState);
            Equal(expected := ActuatorState#MoveToWorkPosition2, actual := _actuator.GetState());

            _cmd := _actuator.GoToWorkPosition2();
            _plcOpenState := Await(_cmd);
            AxUnit.Assert.Equal(expected := PlcOpen#Busy, actual := _plcOpenState);
            Equal(expected := ActuatorState#MoveToWorkPosition2, actual := _actuator.GetState());

            _cmd := _actuator.GoToWorkPosition2();
            _plcOpenState := Await(_cmd);
            AxUnit.Assert.Equal(expected := PlcOpen#Busy, actual := _plcOpenState);
            Equal(expected := ActuatorState#MoveToWorkPosition2, actual := _actuator.GetState());

            _actuator.I_InWorkPosition2 := _sensorActivated;
            _cmd := _actuator.GoToWorkPosition2();
            Equal(expected := ActuatorState#InWorkPosition2, actual := _actuator.GetState());
            _plcOpenState := Await(_cmd);
            AxUnit.Assert.Equal(expected := PlcOpen#Done, actual := _plcOpenState);
            Equal(expected := ActuatorState#InWorkPosition2, actual := _actuator.GetState());
        END_METHOD

        {Test}
        METHOD PUBLIC Command_MoveToWorkPosition_Interrupted_By_MoveToHomePosition
            VAR
                resultHome, resultWork, resultWork2 : BOOL;
            END_VAR

            _actuator.I_InHomePosition := _sensorNotActivated;
            _actuator.I_InWorkPosition := _sensorNotActivated;
            _actuator.I_InWorkPosition2 := _sensorNotActivated;

            // Start MoveToWorkPosition
            _cmd := _actuator.GoToWorkPosition();
            _plcOpenState := Await(_cmd);

            AxUnit.Assert.Equal(expected := PlcOpen#Busy, actual := _plcOpenState);
            Equal(expected := ActuatorState#MoveToWorkPosition, actual := _actuator.GetState());

            ActuatorMoveToHomePos.WriteCyclic(Q => resultHome);
            ActuatorMoveToWorkPos.WriteCyclic(Q => resultWork);
            ActuatorMoveToWorkPos2.WriteCyclic(Q => resultWork2);
            IsFalse(condition := resultHome);
            IsTrue(condition := resultWork);
            IsFalse(condition := resultWork2);

            // Interrupt with MoveToHomePosition
            _cmd := _actuator.GoToHomePosition();
            _plcOpenState := Await(_cmd);

            AxUnit.Assert.Equal(expected := PlcOpen#Busy, actual := _plcOpenState);
            Equal(expected := ActuatorState#MoveToHomePosition, actual := _actuator.GetState());

            ActuatorMoveToHomePos.WriteCyclic(Q => resultHome);
            ActuatorMoveToWorkPos.WriteCyclic(Q => resultWork);
            ActuatorMoveToWorkPos2.WriteCyclic(Q => resultWork2);
            IsTrue(condition := resultHome);
            IsFalse(condition := resultWork);
            IsFalse(condition := resultWork2);

            _actuator.I_InHomePosition := _sensorHasReached;
            _plcOpenState := Await(_cmd);
            AxUnit.Assert.Equal(expected := PlcOpen#Done, actual := _plcOpenState);
            Equal(expected := ActuatorState#InHomePosition, actual := _actuator.GetState());

            // Step 7: Check the actuator outputs again.
            ActuatorMoveToHomePos.WriteCyclic(Q => resultHome);
            ActuatorMoveToWorkPos.WriteCyclic(Q => resultWork);
            ActuatorMoveToWorkPos2.WriteCyclic(Q => resultWork2);
            IsFalse(condition := resultHome);
            IsFalse(condition := resultWork);
            IsFalse(condition := resultWork2);
        END_METHOD

        {Test}
        METHOD PUBLIC Command_MoveToHomePosition_Interrupted_By_MoveToWorkPosition
            VAR
                resultHome, resultWork, resultWork2 : BOOL;
            END_VAR

            _actuator.I_InHomePosition := _sensorNotActivated;
            _actuator.I_InWorkPosition := _sensorNotActivated;
            _actuator.I_InWorkPosition2 := _sensorNotActivated;

            // Start MoveToHomePosition
            _cmd := _actuator.GoToHomePosition();
            _plcOpenState := Await(_cmd);

            AxUnit.Assert.Equal(expected := PlcOpen#Busy, actual := _plcOpenState);
            Equal(expected := ActuatorState#MoveToHomePosition, actual := _actuator.GetState());

            ActuatorMoveToHomePos.WriteCyclic(Q => resultHome);
            ActuatorMoveToWorkPos.WriteCyclic(Q => resultWork);
            ActuatorMoveToWorkPos2.WriteCyclic(Q => resultWork2);
            IsTrue(condition := resultHome);
            IsFalse(condition := resultWork);
            IsFalse(condition := resultWork2);

            // Interrupt with MoveToWorkPosition
            _cmd := _actuator.GoToWorkPosition();
            _plcOpenState := Await(_cmd);

            AxUnit.Assert.Equal(expected := PlcOpen#Busy, actual := _plcOpenState);
            Equal(expected := ActuatorState#MoveToWorkPosition, actual := _actuator.GetState());

            ActuatorMoveToHomePos.WriteCyclic(Q => resultHome);
            ActuatorMoveToWorkPos.WriteCyclic(Q => resultWork);
            ActuatorMoveToWorkPos2.WriteCyclic(Q => resultWork2);
            IsFalse(condition := resultHome);
            IsTrue(condition := resultWork);
            IsFalse(condition := resultWork2);

            _actuator.I_InWorkPosition := _sensorHasReached;
            _plcOpenState := Await(_cmd);
            AxUnit.Assert.Equal(expected := PlcOpen#Done, actual := _plcOpenState);
            Equal(expected := ActuatorState#InWorkPosition, actual := _actuator.GetState());

            ActuatorMoveToHomePos.WriteCyclic(Q => resultHome);
            ActuatorMoveToWorkPos.WriteCyclic(Q => resultWork);
            ActuatorMoveToWorkPos2.WriteCyclic(Q => resultWork2);
            IsFalse(condition := resultHome);
            IsFalse(condition := resultWork);
            IsFalse(condition := resultWork2);
        END_METHOD

        {Test}
        METHOD PUBLIC Command_MoveToWorkPosition2_Interrupted_By_MoveToHomePosition
            VAR
                resultHome, resultWork, resultWork2 : BOOL;
            END_VAR

            // Step 1: Set initial sensor states to indicate the actuator is not in any position.
            _actuator.I_InHomePosition := _sensorNotActivated;
            _actuator.I_InWorkPosition := _sensorNotActivated;
            _actuator.I_InWorkPosition2 := _sensorNotActivated;

            // Step 2: Start MoveToWorkPosition2.
            _cmd := _actuator.GoToWorkPosition2();
            _plcOpenState := Await(_cmd);

            // Step 3: Verify the actuator is in the MoveToWorkPosition2 state.
            AxUnit.Assert.Equal(expected := PlcOpen#Busy, actual := _plcOpenState);
            Equal(expected := ActuatorState#MoveToWorkPosition2, actual := _actuator.GetState());

            // Step 4: Check the actuator outputs.
            ActuatorMoveToHomePos.WriteCyclic(Q => resultHome);
            ActuatorMoveToWorkPos.WriteCyclic(Q => resultWork);
            ActuatorMoveToWorkPos2.WriteCyclic(Q => resultWork2);
            IsFalse(condition := resultHome);
            IsFalse(condition := resultWork);
            IsTrue(condition := resultWork2);

            // Step 5: Interrupt with MoveToHomePosition.
            _cmd := _actuator.GoToHomePosition();
            _plcOpenState := Await(_cmd);

            // Step 6: Verify the actuator is in the MoveToHomePosition state.
            AxUnit.Assert.Equal(expected := PlcOpen#Busy, actual := _plcOpenState);
            Equal(expected := ActuatorState#MoveToHomePosition, actual := _actuator.GetState());

            // Step 7: Check the actuator outputs.
            ActuatorMoveToHomePos.WriteCyclic(Q => resultHome);
            ActuatorMoveToWorkPos.WriteCyclic(Q => resultWork);
            ActuatorMoveToWorkPos2.WriteCyclic(Q => resultWork2);
            IsTrue(condition := resultHome);
            IsFalse(condition := resultWork);
            IsFalse(condition := resultWork2);

            // Step 8: Simulate reaching the home position.
            _actuator.I_InHomePosition := _sensorHasReached;
            _plcOpenState := Await(_cmd);

            // Step 9: Verify the actuator has reached the home position.
            AxUnit.Assert.Equal(expected := PlcOpen#Done, actual := _plcOpenState);
            Equal(expected := ActuatorState#InHomePosition, actual := _actuator.GetState());

            ActuatorMoveToHomePos.WriteCyclic(Q => resultHome);
            ActuatorMoveToWorkPos.WriteCyclic(Q => resultWork);
            ActuatorMoveToWorkPos2.WriteCyclic(Q => resultWork2);
            IsFalse(condition := resultHome);
            IsFalse(condition := resultWork);
            IsFalse(condition := resultWork2);
        END_METHOD

        {Test}
        METHOD PUBLIC Command_MoveToWorkPosition2_Interrupted_By_MoveToWorkPosition
            VAR
                resultHome, resultWork, resultWork2 : BOOL;
            END_VAR

            _actuator.I_InHomePosition := _sensorNotActivated;
            _actuator.I_InWorkPosition := _sensorNotActivated;
            _actuator.I_InWorkPosition2 := _sensorNotActivated;

            // Start MoveToWorkPosition2
            _cmd := _actuator.GoToWorkPosition2();
            _plcOpenState := Await(_cmd);

            AxUnit.Assert.Equal(expected := PlcOpen#Busy, actual := _plcOpenState);
            Equal(expected := ActuatorState#MoveToWorkPosition2, actual := _actuator.GetState());

            ActuatorMoveToHomePos.WriteCyclic(Q => resultHome);
            ActuatorMoveToWorkPos.WriteCyclic(Q => resultWork);
            ActuatorMoveToWorkPos2.WriteCyclic(Q => resultWork2);
            IsFalse(condition := resultHome);
            IsFalse(condition := resultWork);
            IsTrue(condition := resultWork2);

            // Interrupt with MoveToWorkPosition
            _cmd := _actuator.GoToWorkPosition();
            _plcOpenState := Await(_cmd);

            AxUnit.Assert.Equal(expected := PlcOpen#Busy, actual := _plcOpenState);
            Equal(expected := ActuatorState#MoveToWorkPosition, actual := _actuator.GetState());

            ActuatorMoveToHomePos.WriteCyclic(Q => resultHome);
            ActuatorMoveToWorkPos.WriteCyclic(Q => resultWork);
            ActuatorMoveToWorkPos2.WriteCyclic(Q => resultWork2);
            IsFalse(condition := resultHome);
            IsTrue(condition := resultWork);
            IsFalse(condition := resultWork2);

            _actuator.I_InWorkPosition := _sensorHasReached;
            _plcOpenState := Await(_cmd);
            AxUnit.Assert.Equal(expected := PlcOpen#Done, actual := _plcOpenState);
            Equal(expected := ActuatorState#InWorkPosition, actual := _actuator.GetState());

            ActuatorMoveToHomePos.WriteCyclic(Q => resultHome);
            ActuatorMoveToWorkPos.WriteCyclic(Q => resultWork);
            ActuatorMoveToWorkPos2.WriteCyclic(Q => resultWork2);
            IsFalse(condition := resultHome);
            IsFalse(condition := resultWork);
            IsFalse(condition := resultWork2);
        END_METHOD
    END_CLASS

END_NAMESPACE

(* ---- TestActuator3WayErrorHandling.st ---- *)
USING AxUnit.Assert;
USING Simatic.Ax.Commands;

NAMESPACE Simatic.Ax.Actuators

    {TestFixture}
    // Test class for the Actuator2Way class.
    // This class contains tests to verify the behavior of the Actuator2Way component.
    CLASS TestActuator3WayErrorHandling
        VAR
            // Instance of Actuator2Way for testing.
            _actuator, _actuatorStateless : Actuator3Way;

            // Command interface for actuator operations.
            _cmd : itfCommand;

            // State of the PLCOpen command.
            _plcOpenState : PlcOpen;

            // Mock sensors for testing actuator behavior.
            _sensorActivated : EndSwitchMockActivated;
            _sensorNotActivated : EndSwitchMockNotActivated;
            _sensorHasReached : EndSwitchMockHasReached;
            _sensorHasLeft : EndSwitchMockHasLeft;
            _sensorTimeHasElapsed : EndSwitchMockTimeHasElapsed;

            // Actuator Controls
            ActuatorMoveToHomePos : PositionControl;
            ActuatorMoveToWorkPos : PositionControl;
        END_VAR

        {TestSetup}
        // Sets up the test environment by initializing the actuator instance and assigning mock sensors and controls.
        METHOD PUBLIC Setup
            _actuator := _actuatorStateless;
            _actuator.Q_ToHomePosition := ActuatorMoveToHomePos;
            _actuator.Q_ToWorkPosition := ActuatorMoveToWorkPos;
            _actuator.I_InWorkPosition := _sensorNotActivated;
            _actuator.I_InHomePosition := _sensorNotActivated;
        END_METHOD

        {Test}
        // Tests the transition to MoveToWorkPosition state when not in the work position.
        METHOD PUBLIC Command_MoveToWorkPosition_Error_When_Sensor_Time_Has_Elapsed
            VAR
                resultHome, resultWork : BOOL;
            END_VAR

            // Step 1: Set initial sensor states to indicate the actuator is not in any position.
            _actuator.I_InHomePosition := _sensorNotActivated;
            _actuator.I_InWorkPosition := _sensorNotActivated;

            // Step 2: Issue the command to move to work position.
            _cmd := _actuator.GoToWorkPosition();
            _plcOpenState := Await(_cmd);

            // Step 3: Verify the actuator is in the MoveToWorkPosition state.
            Equal(expected := PlcOpen#Busy, actual := _plcOpenState);
            Equal(expected := ActuatorState#MoveToWorkPosition, actual := _actuator.GetState());

            // Step 4: Check the actuator outputs.
            ActuatorMoveToHomePos.WriteCyclic(Q => resultHome);
            ActuatorMoveToWorkPos.WriteCyclic(Q => resultWork);
            IsFalse(condition := resultHome);
            IsTrue(condition := resultWork);

            // Step 5: Simulate reaching the work position.
            _actuator.I_InWorkPosition := _sensorTimeHasElapsed;
            _plcOpenState := Await(_cmd);

            // Step 6: Verify the actuator has reached the work position.
            Equal(expected := PlcOpen#Error, actual := _plcOpenState);
            Equal(expected := ActuatorState#Error, actual := _actuator.GetState());

            // Step 7: Check the actuator outputs again.
            ActuatorMoveToHomePos.WriteCyclic(Q => resultHome);
            ActuatorMoveToWorkPos.WriteCyclic(Q => resultWork);
            IsFalse(condition := resultHome);
            IsFalse(condition := resultWork);
        END_METHOD

        {Test}
        // Tests the transition to MoveToHomePosition state when not in the home position.
        METHOD PUBLIC Reset_Actuator_Returns
            VAR
                resultHome, resultWork : BOOL;
            END_VAR
            THIS.Command_MoveToWorkPosition_Error_When_Sensor_Time_Has_Elapsed();
            // Step 1: Reset Actuator

            _actuator.Reset();

            // Step 2: Verify the actuator is in the MoveToHomePosition state.
            Equal(expected := ActuatorState#Undefined, actual := _actuator.GetState());

            // Step 3: Check the actuator outputs again.
            ActuatorMoveToHomePos.WriteCyclic(Q => resultHome);
            ActuatorMoveToWorkPos.WriteCyclic(Q => resultWork);
            IsFalse(condition := resultHome);
            IsFalse(condition := resultWork);
        END_METHOD

        {Test}
        // Tests the transition to MoveToWorkPosition state when not in the work position.
        METHOD PUBLIC Both_sensors_Active_Retrurs_Error
            VAR
                resultHome, resultWork : BOOL;
            END_VAR

            // Step 1: Set initial sensor states to indicate the actuator is not in any position.
            _actuator.I_InHomePosition := _sensorActivated;
            _actuator.I_InWorkPosition := _sensorActivated;

            // Step 2: Issue the command to move to work position.
            _cmd := _actuator.GoToWorkPosition();
            _plcOpenState := Await(_cmd);

            // Step 3: Verify the actuator is in the MoveToWorkPosition state.
            Equal(expected := PlcOpen#Error, actual := _plcOpenState);
            Equal(expected := ActuatorState#Error, actual := _actuator.GetState());

            // Step 4: Check the actuator outputs again.
            ActuatorMoveToHomePos.WriteCyclic(Q => resultHome);
            ActuatorMoveToWorkPos.WriteCyclic(Q => resultWork);
            IsFalse(condition := resultHome);
            IsFalse(condition := resultWork);
        END_METHOD
    END_CLASS

END_NAMESPACE

(* ---- TestActuator3WayTransitions.st ---- *)
USING AxUnit.Assert;
USING Simatic.Ax.Commands;

NAMESPACE Simatic.Ax.Actuators

    /// Test class for the 3-way actuator transitions.
    /// Input: None.
    /// Returns: None.
    {TestFixture}
    // Test class for the 3-way actuator transitions.
    CLASS TestActuator3WayTransitions
        VAR
            // Instance of Actuator3Way for testing.
            _actuator, _actuatorStateless : Actuator3Way;

            // Stateless instance of Actuator3Way for reinitialization.

            // Mock sensors for testing actuator behavior.
            SensorInHomePosition, _sensorInHomePositionStateless : BooleanEndswitch;
            SensorInWorkPosition, _sensorInWorkPositionStateless : BooleanEndswitch;
            SensorInWorkPosition2, _sensorInWorkPosition2Stateless : BooleanEndswitch;

            // Actuator Controls
            ActuatorMoveToHomePos, _actuatorMoveToHomePosStateless : PositionControl;
            ActuatorMoveToWorkPos, _actuatorMoveToWorkPosStateless : PositionControl;
            ActuatorMoveToWorkPos2, _actuatorMoveToWorkPos2Stateless : PositionControl;

            // Command interface for actuator operations.
            _cmd : itfCommand;
            _plcOpenState : PlcOpen;

        END_VAR
        /// Sets up the test environment for each test.
        /// Input: None.
        /// Returns: None.
        {TestSetup}
        // Sets up the test environment.
        METHOD PUBLIC Setup
            // Reinitialize the actuator instance with a stateless instance.
            _actuator := _actuatorStateless;

            // Assign stateless instances to sensors
            SensorInHomePosition := _sensorInHomePositionStateless;
            SensorInWorkPosition := _sensorInWorkPositionStateless;
            SensorInWorkPosition2 := _sensorInWorkPosition2Stateless;

            // Reinitialize actuator controls
            ActuatorMoveToHomePos := _actuatorMoveToHomePosStateless;
            ActuatorMoveToWorkPos := _actuatorMoveToWorkPosStateless;
            ActuatorMoveToWorkPos2 := _actuatorMoveToWorkPos2Stateless;

            _actuator.Q_ToHomePosition := ActuatorMoveToHomePos;
            _actuator.Q_ToWorkPosition := ActuatorMoveToWorkPos;
            _actuator.Q_ToWorkPosition2 := ActuatorMoveToWorkPos2;

            // Configure end switches
            _actuator.I_InHomePosition := SensorInHomePosition;
            _actuator.I_InWorkPosition := SensorInWorkPosition;
        END_METHOD

        {Test}
        /// Verifies the sequence of end switch states during the MoveToWorkPosition command.
        /// Input: None.
        /// Returns: None.
        METHOD PUBLIC TestMoveToWorkPosition_EndSwitchGoesToZero
            VAR
                q_ToHome, q_ToWork, q_ToWork2 : BOOL;
            END_VAR

            // Step 1: Set initial sensor states.
            SensorInHomePosition.Update(signal := TRUE); // HomePosition starts as true.
            SensorInWorkPosition.Update(signal := FALSE);
            SensorInWorkPosition2.Update(signal := FALSE);

            // Step 2: Issue the command to move to work position.
            _cmd := _actuator.GoToWorkPosition();
            _plcOpenState := Await(_cmd);

            // Step 3: Verify HomePosition becomes false when the actuator starts.
            SensorInHomePosition.Update(signal := FALSE);
            _plcOpenState := Await(_cmd);

            ActuatorMoveToHomePos.WriteCyclic(Q => q_ToHome);
            ActuatorMoveToWorkPos.WriteCyclic(Q => q_ToWork);
            ActuatorMoveToWorkPos2.WriteCyclic(Q => q_ToWork2);

            IsFalse(condition := q_ToHome); // HomePosition is now false.
            IsTrue(condition := q_ToWork);
            IsFalse(condition := q_ToWork2);

            // Step 4: Simulate reaching the work position and verify WorkPosition becomes true.
            SensorInWorkPosition.Update(signal := TRUE);
            _plcOpenState := Await(_cmd);

            ActuatorMoveToHomePos.WriteCyclic(Q => q_ToHome);
            ActuatorMoveToWorkPos.WriteCyclic(Q => q_ToWork);
            ActuatorMoveToWorkPos2.WriteCyclic(Q => q_ToWork2);

            IsFalse(condition := q_ToHome);
            IsFalse(condition := q_ToWork); // WorkPosition is now true.
            IsFalse(condition := q_ToWork2);
        END_METHOD
    END_CLASS

END_NAMESPACE

(* ---- TestEndswitch.st ---- *)
USING Simatic.Ax;
USING AxUnit.Assert;
USING AxUnit.ResultFunctions;
USING System.Strings;
USING Simatic.Ax.Mocks;
USING AxUnit.Mocking;

NAMESPACE Simatic.Ax.Test

    {TestFixture}
    CLASS TestEndswitch

        VAR PROTECTED
            //o : <test instance>; //your test instance
        END_VAR

        METHOD PUBLIC MyMethod
             // write your test code here
            ;
        END_METHOD
    END_CLASS
END_NAMESPACE
NAMESPACE Simatic.Ax.Actuators

    {TestFixture}
    CLASS TestEndswitch
        VAR
            _endswitch, _endswitchStateless  : BooleanEndswitch;
            res : BOOL;
        END_VAR

        {Setup}
        METHOD PUBLIC Setup
            _endswitch := _endswitchStateless;
        END_METHOD

        {Test}
        METHOD PUBLIC TestIsActivated
            VAR
                signal : BOOL := TRUE;
                valid : BOOL := TRUE;
            END_VAR

            _endswitch.Update(signal := TRUE, valid := valid);
            IsTrue(condition := _endswitch.IsActivated());
        END_METHOD

        {Test}
        METHOD PUBLIC TestHasReached
            VAR
                signal : BOOL := TRUE;
                valid : BOOL := TRUE;
            END_VAR

            _endswitch.Update(signal := FALSE, valid := valid);
            _endswitch.Update(signal := TRUE, valid := valid);
            IsTrue(condition := _endswitch.HasReached());
        END_METHOD

        {Test}
        METHOD PUBLIC TestHasLeft
            VAR
                signal : BOOL;
                valid : BOOL := TRUE;
            END_VAR

            _endswitch.Update(signal := TRUE, valid := valid);
            _endswitch.Update(signal := FALSE, valid := valid);
            IsTrue(condition := _endswitch.HasLeft());
        END_METHOD

        {Test}
        METHOD PUBLIC TestEnableSupervision
            VAR
                mode : SuperVisionMode;
            END_VAR

            // Test enabling supervision with different modes
            mode := SuperVisionMode#None;
            _endswitch.EnableSupervision(Mode := mode);
            EqualSuperVisionError(expected := SuperVisionError#None, actual := _endswitch.GetError());

            mode := SuperVisionMode#Reaction;
            _endswitch.EnableSupervision(Mode := mode);
            EqualSuperVisionError(expected := SuperVisionError#None, actual := _endswitch.GetError());

            mode := SuperVisionMode#Action;
            _endswitch.EnableSupervision(Mode := mode);
            EqualSuperVisionError(expected := SuperVisionError#None, actual := _endswitch.GetError());

            mode := SuperVisionMode#PositionControl;
            _endswitch.EnableSupervision(Mode := mode);
            EqualSuperVisionError(expected := SuperVisionError#None, actual := _endswitch.GetError());
        END_METHOD

        {Test}
        METHOD PUBLIC TestUpdateAndCheck
            VAR
                signal : BOOL;
                valid : BOOL := TRUE;
                default : BOOL := FALSE;
            END_VAR

            // Test updating the endswitch with valid signals
            signal := TRUE;
            _endswitch.Update(signal := signal, valid := valid, default := default);
            IsTrue(condition := _endswitch.IsActivated());

            signal := FALSE;
            _endswitch.Update(signal := signal, valid := valid, default := default);
            IsFalse(condition := _endswitch.IsActivated());

            // Test supervision errors
            _endswitch.EnableSupervision(Mode := SuperVisionMode#Reaction);
            _endswitch.Update(signal := FALSE, valid := valid, default := default);
            _endswitch.Update(signal := TRUE, valid := valid, default := default);
            IsTrue(condition := _endswitch.HasReached());

            _endswitch.EnableSuperVision(Mode := SuperVisionMode#Action);
            _endswitch.Update(signal := TRUE, valid := valid, default := default);
            _endswitch.Update(signal := FALSE, valid := valid, default := default);
            IsTrue(condition := _endswitch.HasLeft());
        END_METHOD

        {Test}
        METHOD PUBLIC TestGetError
            VAR
                mode : SuperVisionMode;
            END_VAR

            // Test getting error states
            mode := SuperVisionMode#None;
            _endswitch.EnableSupervision(Mode := mode);
            EqualSuperVisionError(expected := SuperVisionError#None, actual := _endswitch.GetError());

            mode := SuperVisionMode#Reaction;
            _endswitch.EnableSupervision(Mode := mode);
            _endswitch.Update(signal := FALSE);
            _endswitch.Update(signal := TRUE);
            EqualSuperVisionError(expected := SuperVisionError#None, actual := _endswitch.GetError());

            mode := SuperVisionMode#Action;
            _endswitch.EnableSupervision(Mode := mode);
            _endswitch.Update(signal := TRUE);
            _endswitch.Update(signal := FALSE);
            EqualSuperVisionError(expected := SuperVisionError#None, actual := _endswitch.GetError());
        END_METHOD

        {Test}
        // Tests the error behavior for SuperVisionMode#Reaction.
        METHOD PUBLIC Test_ReactionError_Without_any_error
            // Step 1: Mock the OnDelay timer to simulate the timer not elapsed
            AxUnit.Mocking.Mock('System.Timer.OnDelay', 'Simatic.Ax.Mocks.OnDelayMock_false');

            // Step 2: Enable Reaction supervision mode.
            _endswitch.EnableSupervision(Mode := SuperVisionMode#Reaction);

            // Step 3: Simulate the condition where the target position is not reached.
            _endswitch.Update(signal := FALSE);
            _endswitch.Update(signal := FALSE);

            // Step 4: Verify that the no error is returned.
            Equal(expected := SuperVisionError#Evaluating, actual := _endswitch.GetError());

            // Step 5: Simulate the condition where the target position is reached.
            _endswitch.Update(signal := TRUE);

            // Step 6: Verify that the no error is returned.
            Equal(expected := SuperVisionError#None, actual := _endswitch.GetError());
        END_METHOD

        {Test}
        // Tests the error behavior for SuperVisionMode#Reaction.
        METHOD PUBLIC Test_ReactionError_With_error
            // Step 1: Mock the OnDelay timer to simulate the timer not elapsed
            AxUnit.Mocking.Mock('System.Timer.OnDelay', 'Simatic.Ax.Mocks.OnDelayMock_false');

            // Step 2: Enable Reaction supervision mode.
            _endswitch.EnableSupervision(Mode := SuperVisionMode#Reaction);

            // Step 3: Simulate the condition where the target position is not reached.
            _endswitch.Update(signal := FALSE);

            // Step 4: Mock the OnDelay timer to simulate the timer elapsing.
            AxUnit.Mocking.Mock('System.Timer.OnDelay', 'Simatic.Ax.Mocks.OnDelayMock_true');

            // Step 5: Simulate the condition where the target position is not reached.
            _endswitch.Update(signal := FALSE);

            // Step 6: Verify that the ReactionError is returned.
            Equal(expected := SuperVisionError#ReactionError, actual := _endswitch.GetError());
        END_METHOD

        {Test}
        // Tests the error behavior for SuperVisionMode#Action.
        METHOD PUBLIC Test_ActionError_Without_any_error
            // Step 1: Mock the OnDelay timer to simulate the timer not elapsed
            AxUnit.Mocking.Mock('System.Timer.OnDelay', 'Simatic.Ax.Mocks.OnDelayMock_false');

            // Step 2: Enable Reaction supervision mode.
            _endswitch.EnableSupervision(Mode := SuperVisionMode#Action);

            // Step 3: Simulate the condition where the target position is not reached.
            _endswitch.Update(signal := TRUE);
            _endswitch.Update(signal := TRUE);

            // Step 4: Verify that the no error is returned.
            Equal(expected := SuperVisionError#Evaluating, actual := _endswitch.GetError());

            // Step 5: Simulate the condition where the target position is reached.
            _endswitch.Update(signal := FALSE);

            // Step 6: Verify that the no error is returned.
            Equal(expected := SuperVisionError#None, actual := _endswitch.GetError());

        END_METHOD

        {Test}
        // Tests the error behavior for SuperVisionMode#Action.
        METHOD PUBLIC Test_ActionError_With_error
            // Step 1: Mock the OnDelay timer to simulate the timer not elapsed
            AxUnit.Mocking.Mock('System.Timer.OnDelay', 'Simatic.Ax.Mocks.OnDelayMock_false');

            // Step 2: Enable Reaction supervision mode.
            _endswitch.EnableSupervision(Mode := SuperVisionMode#Action);

            // Step 3: Simulate the condition where the target position is not reached.
            _endswitch.Update(signal := FALSE);

            // Step 4: Mock the OnDelay timer to simulate the timer elapsing.
            AxUnit.Mocking.Mock('System.Timer.OnDelay', 'Simatic.Ax.Mocks.OnDelayMock_true');

            // Step 5: Simulate the condition where the target position is not reached.
            _endswitch.Update(signal := FALSE);

            // Step 6: Verify that the ReactionError is returned.
            Equal(expected := SuperVisionError#ActionError, actual := _endswitch.GetError());
        END_METHOD

        {Test}
        // Tests the error behavior for SuperVisionMode#PositionControl.
        METHOD PUBLIC Test_Error_Behavior_PositionControl
            // Step 1: Enable PositionControl supervision mode.
            _endswitch.EnableSupervision(Mode := SuperVisionMode#PositionControl);

            // Step 2: Simulate an unexpected position change.
            _endswitch.Update(signal := TRUE);
            _endswitch.Update(signal := FALSE);

            // Step 3: Verify that the PositionError is returned.
            Equal(expected := SuperVisionError#PositionError, actual := _endswitch.GetError());
        END_METHOD

        {Test}
        // Tests the Evaluating state for SuperVisionMode#Reaction.
        METHOD PUBLIC Test_Evaluating_State_Reaction
            // Step 1: Enable Reaction supervision mode.
            _endswitch.EnableSupervision(Mode := SuperVisionMode#Reaction);

            // Step 2: Simulate the condition where the target position is not yet reached.
            _endswitch.Update(signal := FALSE);

            // Step 3: Verify that the Evaluating state is returned.
            Equal(expected := SuperVisionError#Evaluating, actual := _endswitch.GetError());
        END_METHOD

        {Test}
        // Tests the Evaluating state for SuperVisionMode#Action.
        METHOD PUBLIC Test_Evaluating_State_Action
            // Step 1: Enable Action supervision mode.
            _endswitch.EnableSupervision(Mode := SuperVisionMode#Action);

            // Step 2: Simulate the condition where no action has occurred yet.
            _endswitch.Update(signal := TRUE);

            // Step 3: Verify that the Evaluating state is returned.
            Equal(expected := SuperVisionError#Evaluating, actual := _endswitch.GetError());
        END_METHOD

        {Test}
        // Tests the Evaluating state for SuperVisionMode#PositionControl.
        METHOD PUBLIC Test_Evaluating_State_PositionControl
            // Step 1: Enable PositionControl supervision mode.
            _endswitch.EnableSupervision(Mode := SuperVisionMode#PositionControl);

            // Step 2: Simulate the condition where no unexpected position change has occurred yet.
            _endswitch.Update(signal := TRUE);

            // Step 3: Verify that the Evaluating state is returned.
            Equal(expected := SuperVisionError#Evaluating, actual := _endswitch.GetError());
        END_METHOD
    END_CLASS

    FUNCTION EqualSuperVisionError
        VAR_INPUT
            expected : SuperVisionError;
            actual : SuperVisionError;
            messageOnFail : STRING;
            {CallerFilePath}
            file : WSTRING[1024];
            {CallerLineNumber}
            line : INT;
        END_VAR
        VAR_TEMP
            messageStr : STRING;
        END_VAR

        IF expected = actual THEN
            axunit_Succeed();
        ELSE
            messageStr := Concat('Expected = ', ToStringSuperVisionError(expected), ' Actual = ', ToStringSuperVisionError(actual));
            axunit_Fail(messageStr, file, line);
        END_IF;
    END_FUNCTION

    FUNCTION ToStringSuperVisionError : STRING
        VAR_INPUT
            val : SuperVisionError;
        END_VAR
        IF val = SuperVisionError#None THEN
            ToStringSuperVisionError := 'None';
        ELSIF val = SuperVisionError#PositionError THEN
            ToStringSuperVisionError := 'PositionControl';
        ELSIF val = SuperVisionError#ActionError THEN
            ToStringSuperVisionError := 'Action';
        ELSIF val = SuperVisionError#ReactionError THEN
            ToStringSuperVisionError := 'Reaction';
        ELSE
            ToStringSuperVisionError := 'Unknown';
        END_IF;
    END_FUNCTION

END_NAMESPACE

(* ---- TestPositionControl.st ---- *)
USING AxUnit.Assert;
USING Simatic.Ax.Actuators;

NAMESPACE Simatic.Ax.Actuators.Tests

    /// Test fixture for PositionControl class functionality.
    {TestFixture}
    CLASS TestPositionControl
        VAR
            /// Instance of PositionControl for testing.
            _positionControl, _positionControlStateless : PositionControl;

            /// Result variables for testing.
            _result : BOOL;
            _output : BOOL;
        END_VAR

        {TestSetup}
        METHOD PUBLIC TestSetup
            _positionControl := _positionControlStateless;
        END_METHOD

        /// Test that Set method activates the position control.
        {Test}
        METHOD PUBLIC Test_Set_ActivatesPosition
            // Arrange
            _positionControl.Behavior := PositionBehavior#SelfHold;

            // Act
            _result := _positionControl.Set();
            _positionControl.WriteCyclic(Q => _output);

            // Assert
            Equal(expected := TRUE, actual := _result);
            Equal(expected := TRUE, actual := _output);
        END_METHOD

        /// Test that Reset method deactivates the position control.
        {Test}
        METHOD PUBLIC Test_Reset_DeactivatesPosition
            // Arrange
            _positionControl.Set(); // First set it to true

            // Act
            _result := _positionControl.Reset();
            _positionControl.WriteCyclic(Q => _output);

            // Assert
            Equal(expected := FALSE, actual := _result);
            Equal(expected := FALSE, actual := _output);
        END_METHOD

        /// Test that Hold method with ActiveHold behavior keeps position active.
        {Test}
        METHOD PUBLIC Test_Hold_ActiveHold_KeepsPositionActive
            // Arrange
            _positionControl.Behavior := PositionBehavior#ActiveHold;

            // Act
            _result := _positionControl.Hold();
            _positionControl.WriteCyclic(Q => _output);

            // Assert
            Equal(expected := TRUE, actual := _result);
            Equal(expected := TRUE, actual := _output);
        END_METHOD

        /// Test that Hold method with SelfHold behavior deactivates position.
        {Test}
        METHOD PUBLIC Test_Hold_SelfHold_DeactivatesPosition
            // Arrange
            _positionControl.Behavior := PositionBehavior#SelfHold;
            _positionControl.Set(); // First set it to true

            // Act
            _result := _positionControl.Hold();
            _positionControl.WriteCyclic(Q => _output);

            // Assert
            Equal(expected := FALSE, actual := _result);
            Equal(expected := FALSE, actual := _output);
        END_METHOD

        /// Test sequence: Set -> Hold (ActiveHold) -> Reset.
        {Test}
        METHOD PUBLIC Test_Sequence_Set_HoldActiveHold_Reset
            // Arrange
            _positionControl.Behavior := PositionBehavior#ActiveHold;

            // Act & Assert - Set
            _result := _positionControl.Set();
            _positionControl.WriteCyclic(Q => _output);
            Equal(expected := TRUE, actual := _result);
            Equal(expected := TRUE, actual := _output);

            // Act & Assert - Hold
            _result := _positionControl.Hold();
            _positionControl.WriteCyclic(Q => _output);
            Equal(expected := TRUE, actual := _result);
            Equal(expected := TRUE, actual := _output);

            // Act & Assert - Reset
            _result := _positionControl.Reset();
            _positionControl.WriteCyclic(Q => _output);
            Equal(expected := FALSE, actual := _result);
            Equal(expected := FALSE, actual := _output);
        END_METHOD

        /// Test sequence: Set -> Hold (SelfHold) -> Set.
        {Test}
        METHOD PUBLIC Test_Sequence_Set_HoldSelfHold_Set
            // Arrange
            _positionControl.Behavior := PositionBehavior#SelfHold;

            // Act & Assert - Set
            _result := _positionControl.Set();
            _positionControl.WriteCyclic(Q => _output);
            Equal(expected := TRUE, actual := _result);
            Equal(expected := TRUE, actual := _output);

            // Act & Assert - Hold (should deactivate)
            _result := _positionControl.Hold();
            _positionControl.WriteCyclic(Q => _output);
            Equal(expected := FALSE, actual := _result);
            Equal(expected := FALSE, actual := _output);

            // Act & Assert - Set again
            _result := _positionControl.Set();
            _positionControl.WriteCyclic(Q => _output);
            Equal(expected := TRUE, actual := _result);
            Equal(expected := TRUE, actual := _output);
        END_METHOD

        /// Test default behavior is SelfHold.
        {Test}
        METHOD PUBLIC Test_DefaultBehavior_IsSelfHold
            // Arrange & Act
            _result := _positionControl.Hold();
            _positionControl.WriteCyclic(Q => _output);

            // Assert
            Equal(expected := FALSE, actual := _result);
            Equal(expected := FALSE, actual := _output);
        END_METHOD

        /// Test changing behavior affects Hold method.
        {Test}
        METHOD PUBLIC Test_ChangingBehavior_AffectsHoldMethod
            // Arrange & Act - SelfHold
            _positionControl.Behavior := PositionBehavior#SelfHold;
            _result := _positionControl.Hold();
            _positionControl.WriteCyclic(Q => _output);

            // Assert - SelfHold
            Equal(expected := FALSE, actual := _result);
            Equal(expected := FALSE, actual := _output);

            // Arrange & Act - ActiveHold
            _positionControl.Behavior := PositionBehavior#ActiveHold;
            _result := _positionControl.Hold();
            _positionControl.WriteCyclic(Q => _output);

            // Assert - ActiveHold
            Equal(expected := TRUE, actual := _result);
            Equal(expected := TRUE, actual := _output);
        END_METHOD
    END_CLASS

    /// Test fixture for NullPositionControl class functionality.
    {TestFixture}
    CLASS TestNullPositionControl
        VAR
            /// Instance of NullPositionControl for testing.
            _nullPositionControl : NullPositionControl;

            /// Result variable for testing.
            _result : BOOL;
        END_VAR

        /// Test that Set method returns default value.
        {Test}
        METHOD PUBLIC Test_Set_ReturnsDefaultValue
            // Act
            _result := _nullPositionControl.Set();

            // Assert
            Equal(expected := FALSE, actual := _result);
        END_METHOD

        /// Test that Reset method returns default value.
        {Test}
        METHOD PUBLIC Test_Reset_ReturnsDefaultValue
            // Act
            _result := _nullPositionControl.Reset();

            // Assert
            Equal(expected := FALSE, actual := _result);
        END_METHOD

        /// Test that Hold method returns default value.
        {Test}
        METHOD PUBLIC Test_Hold_ReturnsDefaultValue
            // Act
            _result := _nullPositionControl.Hold();

            // Assert
            Equal(expected := FALSE, actual := _result);
        END_METHOD
    END_CLASS

END_NAMESPACE

(* ---- TestStateLogger.st ---- *)
USING AxUnit.Assert;
USING System.Strings;
NAMESPACE Simatic.Ax.Actuators

    {TestFixture}
    CLASS TestStateLogger
        VAR
            _o, _oStateLess  : StateLogger;
            _msgBuffer : ARRAY[2..4] OF LogMessage;
        END_VAR

        {TestSetup}
        METHOD PUBLIC Setup
            _o := _oStateLess;
            _o.MsgBuffer := REF(_msgBuffer);
        END_METHOD

        {Test}
        METHOD PUBLIC TestWriteLog
            VAR
                msg : STRING := 'Test message';
                loglevel : LogLevel := LogLevel#Info;
            END_VAR

            _o.SetLogLevel(loglevel := LogLevel.Info);
            _o.WriteLog(msg := msg, loglevel := loglevel);
            IsTrue(condition := _o.MsgBuffer^[2].message = msg);
        END_METHOD

        {Test}
        METHOD PUBLIC TestCircularBuffer
            VAR
                i : DINT;
                msg : STRING;
                loglevel : LogLevel := LogLevel#Info;
            END_VAR

            _o.SetLogLevel(loglevel := loglevel);
            FOR i := 2 TO 4 DO
                msg := CONCAT('Message ', Conversion.Integer.ToString(i));
                _o.WriteLog(msg := msg, loglevel := loglevel);
            END_FOR;
            Equal(actual := _o.MsgBuffer^[2].message, expected := 'Message 2');
            Equal(actual := _o.MsgBuffer^[3].message, expected := 'Message 3');
            Equal(actual := _o.MsgBuffer^[4].message, expected := 'Message 4');
            FOR i := 6 TO 8 DO
                msg := CONCAT('Message ', Conversion.Integer.ToString(i));
                _o.WriteLog(msg := msg, loglevel := loglevel);
            END_FOR;
            Equal(actual := _o.MsgBuffer^[2].message, expected := 'Message 6');
            Equal(actual := _o.MsgBuffer^[3].message, expected := 'Message 7');
            Equal(actual := _o.MsgBuffer^[4].message, expected := 'Message 8');
        END_METHOD
    END_CLASS

END_NAMESPACE
